Fanuc KAREL source: ka00054.KL

-- PROVISIONAL review KL for V1013-1; original PC SHA256 28ca2cb9b4b523761fee1219d2cd869a22af8d90a6d59bf5e61b08cbcf7fd1a4
-- Incomplete behavior may be omitted. Consult companion uncertainty JSON. Do not deploy.
PROGRAM KA00054
%NOLOCKGROUP
-- UNRESOLVED_DECL SRC type=000101
-- UNRESOLVED_DECL DST type=000102
BEGIN
  -- UNRESOLVED_PC offsets 5-25; opcodes 49,7E,4A
  -- UNRESOLVED_PC offsets 30-34; opcodes 7F
END KA00054
